Staubli VAL3: saveApplication.pgx

program saveApplication()
  local num nResult
begin
    //
  //\var nResult
  //
// save the application
  nResult=app:libSave()
  // check if saving was successfull
  if nResult!=0
    popUpMsg("Saving Application failed: "+toString("",nResult))
  else
    SYS:bModified=false
  endIf
  data:libSave()
end
